(* PLC project Generated.project, CODESYS CODESYS V3.5 SP19 Patch 1 *)
(* stored: creationDateTime 2026-10-28T23:07:00.277837, modificationDateTime 2026-10-28T23:07:00.277837 *)

(* ═══════════════════════════════════════════════════════════════ 🧪 FB_Sim_Encoder — Simulation physique d'un codeur absolu de treuil ─────────────────────────────────────────────────────────────── 📄 Doc métier : DOC/AF/AF_Partie-13_Fonction_Simulation_v2.5.md 📄 Spec composant : DOC/AF/AF_Partie-13_Fonction_Simulation/FB_Sim_Encoder_v1.1.md 🧩 Brique réduite (Partie3 §1bis, "briques E/S & diagnostics") : pas de contrat Enable/Reset/Error complet, pas de StartStop/SafeStop — outil de banc, pas du métier machine. 🎯 Rôle : fait "compter" un codeur absolu comme si le treuil tournait réellement, à partir des relais de sens commandés et du palier de vitesse courant. 📥 Enable : simulation active (SimulationModeActive AND NOT BusEncoderMxIsReal) 📥 RelayFwd/RelayRev : sens commandé (contacteurs de sens du treuil) 📥 StepNumber : palier vitesse courant (1..5) — ex. instWinchM1.StepNumber Vitesse = interpolation linéaire : palier 1 → MinSpeedMps (1 m/s), palier 5 → MaxSpeedMps (2 m/s). 📥 PresetCmd : TRUE le cycle où un preset (homing) doit être appliqué (PresettTrigCmd = 2) 📥 PresetValue : valeur brute à charger lors du preset 📥 SpeedScaleFactor : facteur fin de confort (réglable à chaud, sans recompiler). Défaut 1.0 = vitesse réelle telle que définie par MinSpeedMps/MaxSpeedMps/PointsPerRev/CableM_PerRev/CycleTimeS. 📤 RawPosOut : position brute simulée (UDINT), à aiguiller à la place de la valeur EtherCAT réelle quand le device n'est pas Operational (voir PRG_02_Encoders.st) 🔒 Comptage brut : entier SIGNÉ 32 bits (le conteneur UDINT n'est qu'un support d'échange, relu en DINT par toute la chaîne aval). Il franchit 0 sans jamais s'y figer ; la seule borne est la plage de représentation, signalée par CountSaturated — jamais muette. 📤 CountSaturated : comptage en butée de plage du modèle (saturation signalée, vitesse purgée) `RawPos` en `VAR_IN_OUT`, référencé depuis `GVL_PERSISTENT` (même pattern que `Calib` dans `FB_Encoder_Homing`) — `PERSISTENT` n'est valide que sur du `VAR_GLOBAL` en CODESYS, pas sur une variable locale de FB. Un vrai codeur absolu physique conserve son comptage brut même à travers un reset FROID (indépendant de l'automate). ═══════════════════════════════════════════════════════════════ === DECLARATION (à coller dans la partie déclaration du POU FB_Sim_Encoder) === *)
FUNCTION_BLOCK FB_Sim_Encoder
  VAR_INPUT
    Enable : BOOL;  (* --> [CMD] Active la simulation *)
    RelayFwd : BOOL;  (* --> [HW] Sens commandé avant *)
    RelayRev : BOOL;  (* --> [HW] Sens commandé arrière *)
    StepNumber : INT;  (* --> [CMD] Palier vitesse courant (1..5, 0 = arrêt) *)
    PresetCmd : BOOL;  (* --> [CMD] Applique un preset (homing) *)
    PresetValue : UDINT;  (* --> [CFG] Valeur brute à charger au preset *)
    SpeedScaleFactor : REAL := 1;  (* --> [CFG] Facteur fin de confort (défaut 1.0) *)
    CoastDistanceM : REAL := 0;  (* --> [CFG] Distance de roulis inertiel apres coupure des relais (m). 0 = arret net (defaut). >0 = le treuil continue a vitesse palier 1 dans le dernier sens sur CoastDistanceM metres -> modelise l'anticipation d'arret mecanique (ex. benne). *)
    PresetLatencyCycles : INT := 3;  (* --> [CFG] Nb cycles automate avant application du preset (referencement non instantane) *)
    TestOffsetCmd : BOOL;  (* --> [TST] Front montant = applique TestOffsetPts (test banc) *)
    TestOffsetPts : DINT := 0;  (* --> [TST] Décalage signé à appliquer (points bruts) *)
    MinSpeedMps : REAL := 1;  (* 📐 Paramètres physiques du treuil (mêmes valeurs que FB_Encoder_Scale) + vitesse réelle. Vitesse simulée = interpolation linéaire du palier : palier 1 → MinSpeedMps, palier 5 → MaxSpeedMps. --> [CFG] Vitesse palier 1 (m/s) *)
    MaxSpeedMps : REAL := 2;  (* --> [CFG] Vitesse palier 5 (m/s) *)
    PointsPerRev : UDINT := 8192;  (* --> [CFG] Résolution codeur (pts/tour) *)
    CableM_PerRev : REAL := 2;  (* --> [CFG] Développement câble (m/tour) *)
    CycleTimeS : REAL := 0.01;  (* --> [CFG] Période tâche PLC (s) — MainTask 10 ms *)
    SpeedReportTauS : REAL := 0;  (* --> [CFG][SYNTHETIQUE] Constante de temps 1er ordre du retour vitesse *)
    CoastDecelUp_Mps2 : REAL := 1.2;  (* --> [CFG] Deceleration en montee (m/s²) : v0²/(2*0.543m) = 1.20 *)
    CoastDecelDown_Mps2 : REAL := 0.93;  (* --> [CFG] Deceleration en descente (m/s²) : v0²/(2*1.205m) = 0.93 *)
    MechanicStopEngaged : BOOL := FALSE;  (* --> [HW] Butee mecanique engagee (coupe net le glissement) *)
  END_VAR
  VAR_OUTPUT
    RawPosOut : UDINT;  (* <-- [DIAG] Position brute simulée *)
    RawSpdOut : DINT;  (* <-- [DIAG] Vitesse brute simulée (0x6031:01 en 0.1 RPM) *)
    CountSaturated : BOOL;  (* <-- [DIAG] Comptage en butée de plage du modèle (saturation signalée) *)
    CoastActive : BOOL;  (* <-- [DIAG] Indicateur de glissement inertiel en cours (T421) *)
  END_VAR
  VAR_IN_OUT
    RawPos : UDINT;  (* <-> [BUS] Référence _SimEncoderRawPosM1/M2 (survit au reset froid) *)
  END_VAR
  VAR
    Increment : UDINT;  (* . [LOC] Points ajoutés par cycle *)
    EffStep : INT;  (* . [LOC] Pas borné (>= 1) *)
    SpeedMps : REAL;  (* . [LOC] Vitesse simulée (m/s) *)
    TestOffsetEdge : R_TRIG;  (* . [LOC] Front TestOffsetCmd *)
    PresetEdge : R_TRIG;  (* . [LOC] Front montant PresetCmd *)
    PresetPending : BOOL;  (* . [LOC] Preset en attente d'application (latence) *)
    PresetCount : INT;  (* . [LOC] Compteur cycles de latence restants *)
    IncrStep1 : UDINT;  (* . [LOC] Increment par cycle a vitesse palier 1 (pour le roulis) *)
    MovingDir : INT;  (* . [LOC] Dernier sens actif : +1 avant, -1 arriere, 0 arret *)
    CoastPtsLeft : REAL;  (* . [LOC] Roulis inertiel restant (points bruts) *)
    TargetSpeedMps : REAL;  (* . [LOC] Vitesse instantanee signee du modele position, avant filtrage retour *)
    ReportedSpeedMps : REAL;  (* . [LOC] Vitesse rapportee filtree 1er ordre, publiee dans RawSpdOut *)
    CoastSpeedMps : REAL;  (* . [LOC] Vitesse instantanee signee pendant le glissement inertiel (T421) *)
    CST_CountTravelLimitPts : DINT := 1073741824;  (* 🛑 Plage de comptage du modèle : le compteur brut est un entier SIGNÉ 32 bits (le conteneur UDINT n'est qu'un support d'échange, relu en DINT par toute la chaîne aval). La garde reste volontairement à la moitié de la plage signée (2^30 pts = 262 144 m de câble) : inatteignable en essai, elle interdit tout rebouclage silencieux si le modèle consommait toute sa plage. 2^30 pts — demi-plage signée *)
  END_VAR

            

// === IMPLEMENTATION (à coller dans le corps ST du POU FB_Sim_Encoder) ===

{region "§1 Gate"}
IF NOT Enable THEN
    RawPosOut := RawPos;
    // Comptage non evalue hors simulation : la saturation ne doit pas rester figee a TRUE.
    CountSaturated := FALSE;
    RETURN;
END_IF;
{endregion}

{region "§2 Injection test"}
// Injection test banc : VRAI saut de position (comme un glissement réel),
// pour tester Concept 1 / Méca E ET le rattrapage joystick (voir GVL_Simulation bandeau).
TestOffsetEdge(CLK := TestOffsetCmd);
IF TestOffsetEdge.Q THEN
    RawPos := DINT_TO_UDINT(UDINT_TO_DINT(RawPos) + TestOffsetPts);
END_IF;
{endregion}

{region "§3 Comptage"}
// 🎚️ Vitesse simulée = interpolation linéaire du palier (palier 1 → MinSpeedMps, palier 5 → MaxSpeedMps),
// pas par pas de (Max−Min)/4. Palier 0 (arrêt) ramène au palier 1 mais aucun mouvement n'est
// appliqué tant que RelayFwd/RelayRev = FALSE (section plus bas).
EffStep  := MAX(StepNumber, 1);
SpeedMps := MinSpeedMps + (INT_TO_REAL(EffStep) - 1.0) * ((MaxSpeedMps - MinSpeedMps) / 4.0);
// Points par cycle = vitesse (m/s) × points par mètre × période tâche (s) × facteur confort.
Increment := REAL_TO_UDINT(SpeedMps * (UDINT_TO_REAL(PointsPerRev) / CableM_PerRev) * CycleTimeS * SpeedScaleFactor);
// Increment "lent" (palier 1) : vitesse du roulis inertiel apres coupure des relais.
IncrStep1 := REAL_TO_UDINT(MinSpeedMps * (UDINT_TO_REAL(PointsPerRev) / CableM_PerRev) * CycleTimeS * SpeedScaleFactor);

// Front du preset : lance la latence de referencement (le codeur réel n'est pas
// instantane — il met PresetLatencyCycles cycles a se re-referencer apres le front).
PresetEdge(CLK := PresetCmd);
IF PresetEdge.Q THEN
    PresetPending := TRUE;
    PresetCount := PresetLatencyCycles;
END_IF;

// 📐 Le comptage brut est un entier SIGNÉ 32 bits : le conteneur UDINT n'est qu'un support
// d'échange (toute la chaîne aval le relit via UDINT_TO_DINT : FB_Encoder_Scale, FB_Encoder_Homing).
// Sa valeur 0 n'est donc PAS une butée mécanique — c'est un point de passage comme un autre, et
// c'est la seule façon de rester fidèle à un codeur absolu, dont le zéro de comptage est arbitraire.
// Aucune branche de comptage ne borne donc à un littéral : seule la garde de plage §3bis intervient,
// et elle est signalée (CountSaturated).
// Pendant l'attente du preset, la position brute est conservee (le codeur n'a pas encore re-reference).
// Le mouvement est gelé pendant la latence, comme un codeur réel en cours de referencement.
IF PresetPending THEN
    IF PresetCount > 0 THEN
        PresetCount := PresetCount - 1;
    ELSE
        // Latence écoulée : applique la valeur cible du preset.
        RawPos := PresetValue;
        PresetPending := FALSE;
    END_IF;
    TargetSpeedMps := 0.0;
ELSIF RelayFwd AND NOT RelayRev THEN
    IF NOT MechanicStopEngaged THEN
        RawPos := DINT_TO_UDINT(UDINT_TO_DINT(RawPos) + UDINT_TO_DINT(Increment));
        MovingDir := 1;
        CoastSpeedMps := SpeedMps;
        CoastPtsLeft := CoastDistanceM * (UDINT_TO_REAL(PointsPerRev) / CableM_PerRev);
        TargetSpeedMps := SpeedMps;
    ELSE
        MovingDir := 0;
        CoastSpeedMps := 0.0;
        CoastPtsLeft := 0.0;
        TargetSpeedMps := 0.0;
    END_IF;
    CoastActive := FALSE;
ELSIF RelayRev AND NOT RelayFwd THEN
    IF NOT MechanicStopEngaged THEN
        RawPos := DINT_TO_UDINT(UDINT_TO_DINT(RawPos) - UDINT_TO_DINT(Increment));
        MovingDir := -1;
        CoastSpeedMps := -SpeedMps;
        CoastPtsLeft := CoastDistanceM * (UDINT_TO_REAL(PointsPerRev) / CableM_PerRev);
        TargetSpeedMps := -SpeedMps;
    ELSE
        MovingDir := 0;
        CoastSpeedMps := 0.0;
        CoastPtsLeft := 0.0;
        TargetSpeedMps := 0.0;
    END_IF;
    CoastActive := FALSE;
ELSE
    // Relais coupes (ou les deux actifs = conflit) : glissement inertiel (T421)
    IF MechanicStopEngaged THEN
        MovingDir := 0;
        CoastSpeedMps := 0.0;
        CoastPtsLeft := 0.0;
        TargetSpeedMps := 0.0;
        CoastActive := FALSE;
    ELSIF (CoastDistanceM > 0.0) AND (CoastPtsLeft >= 1.0) AND (MovingDir <> 0) THEN
        // Mode historique compatibilite (si CoastDistanceM explicitement configure > 0)
        CoastActive := TRUE;
        IF MovingDir = 1 THEN
            RawPos := DINT_TO_UDINT(UDINT_TO_DINT(RawPos) + UDINT_TO_DINT(IncrStep1));
            TargetSpeedMps := MinSpeedMps;
        ELSE
            RawPos := DINT_TO_UDINT(UDINT_TO_DINT(RawPos) - UDINT_TO_DINT(IncrStep1));
            TargetSpeedMps := -MinSpeedMps;
        END_IF;
        CoastPtsLeft := CoastPtsLeft - UDINT_TO_REAL(IncrStep1);
    ELSIF (ABS(CoastSpeedMps) > 0.005) AND (MovingDir <> 0) THEN
        // 🆕 Modele dynamique continu T421 : deceleration signee continue calee sur trace reelle
        CoastActive := TRUE;
        IF CoastSpeedMps > 0.0 THEN
            CoastSpeedMps := CoastSpeedMps - CoastDecelUp_Mps2 * CycleTimeS;
            IF CoastSpeedMps <= 0.005 THEN
                CoastSpeedMps := 0.0;
                MovingDir := 0;
                CoastActive := FALSE;
            END_IF;
        ELSE
            CoastSpeedMps := CoastSpeedMps + CoastDecelDown_Mps2 * CycleTimeS;
            IF CoastSpeedMps >= -0.005 THEN
                CoastSpeedMps := 0.0;
                MovingDir := 0;
                CoastActive := FALSE;
            END_IF;
        END_IF;

        // Deplacement par cycle correspondant a CoastSpeedMps
        Increment := REAL_TO_UDINT(ABS(CoastSpeedMps) * (UDINT_TO_REAL(PointsPerRev) / CableM_PerRev) * CycleTimeS * SpeedScaleFactor);
        IF CoastSpeedMps > 0.0 THEN
            RawPos := DINT_TO_UDINT(UDINT_TO_DINT(RawPos) + UDINT_TO_DINT(Increment));
            TargetSpeedMps := CoastSpeedMps;
        ELSIF CoastSpeedMps < 0.0 THEN
            RawPos := DINT_TO_UDINT(UDINT_TO_DINT(RawPos) - UDINT_TO_DINT(Increment));
            TargetSpeedMps := CoastSpeedMps;
        ELSE
            TargetSpeedMps := 0.0;
        END_IF;
    ELSE
        MovingDir := 0;
        CoastSpeedMps := 0.0;
        CoastPtsLeft := 0.0;
        TargetSpeedMps := 0.0;
        CoastActive := FALSE;
    END_IF;
END_IF;
{endregion}

{region "§3bis Garde de plage de comptage"}
// 🛑 SEULE borne du comptage : la plage de représentation signée. Elle est SIGNALÉE
// (CountSaturated) et cohérente — une position bornée ne publie plus de vitesse de mouvement,
// ce qui interdit la signature « position figée + vitesse non nulle + zéro défaut ».
CountSaturated := FALSE;
IF UDINT_TO_DINT(RawPos) > CST_CountTravelLimitPts THEN
    RawPos := DINT_TO_UDINT(CST_CountTravelLimitPts);
    CountSaturated := TRUE;
ELSIF UDINT_TO_DINT(RawPos) < -CST_CountTravelLimitPts THEN
    RawPos := DINT_TO_UDINT(-CST_CountTravelLimitPts);
    CountSaturated := TRUE;
END_IF;
IF CountSaturated THEN
    TargetSpeedMps := 0.0;
END_IF;
{endregion}

{region "§4 Sortie"}
RawPosOut := RawPos;
// Retour vitesse rapporte (RawSpdOut) : 1er ordre vers TargetSpeedMps. SpeedReportTauS=0.0
// -> alpha=1 -> saut instantane (comportement historique inchange).
ReportedSpeedMps := ReportedSpeedMps
    + (CycleTimeS / (SpeedReportTauS + CycleTimeS)) * (TargetSpeedMps - ReportedSpeedMps);
// Formule inverse vitesse brute EtherCAT CoE (0.1 RPM) :
// SpdValue = (V_mps * 60.0) / (0.1 * CableM_PerRev) = V_mps * 300.0 (sur tambour 2m)
IF (CableM_PerRev > 0.0) THEN
    RawSpdOut := REAL_TO_DINT((ReportedSpeedMps * 60.0) / (0.1 * CableM_PerRev) * SpeedScaleFactor);
ELSE
    RawSpdOut := 0;
END_IF;
{endregion}

          
END_FUNCTION_BLOCK
